RoboDK station: Example-01.a-Robot Painting - Universal Robots.rdk

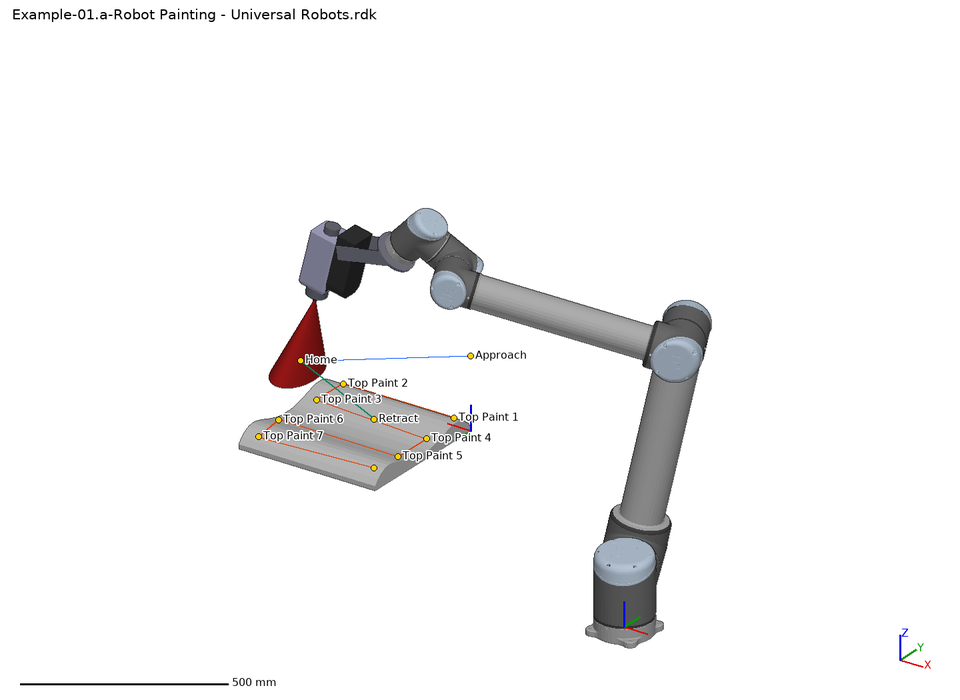
[picture v0: the station drawn from its stored meshes, robots at their saved joint values, targets as dots, program paths as lines]
Station Painting-Tutorial. Poses are relative to the parent item; angles as X-Y-Z fixed-axis rotations.
  - frame UR10 Base at (0, 0, 0) mm
    - robot UR10: 6 axes, payload 10 kg, reach 1300 mm, repeatability 0.1 mm, weight 28.9 kg
        modified DH rows (alpha deg, a mm, theta deg, d mm): 0, 0, 0, 118; 90, 0, 180, 0; 0, 612.7, 0, 0; 0, 571.6, 0, 163.9; -90, 0, 0, 115.7; 90, 0, 180, 92.2
        joint limits [-360, -360, -360, -360, -360, -360] to [360, 360, 360, 360, 360, 360]; home [0, -90, 90, 0, 90, 0]; saved at [-151.986, -78.222, -86.642, -64.602, 73.062, 110.032]
      - tool Paint gun, TCP at (50, 0, 450) mm, rotated rx 0 ry 30 rz 0 deg, size 203.2 x 279.7 x 471.5 mm
    - frame Frame 2 at (-800, 500, 100) mm, rotated rx 0 ry 0 rz 180 deg
      - object Object Inspection at (0, 0, 0) mm, size 400 x 400 x 46.2 mm, geometry from Object Inspection.stp
      - target Home (Cartesian target) at (66.76, 615.12, 413.71) mm, rotated rx 179.14 ry 13.35 rz -178.18 deg; joints [-151.986, -78.222, -86.642, -64.602, 73.062, 110.032] of UR10
      - target Approach (Cartesian target) at (0, 0, 200) mm, rotated rx 180 ry 0 rz 180 deg; joints [-208.691, -96.314, -82.153, -64.673, 103.889, 64.641] of UR10
      - target Top Paint 1 (Cartesian target) at (31.07, 24.78, 35.36) mm, rotated rx 143.81 ry -11.15 rz 165.19 deg; joints [-219.536, -114.993, -76.946, -70.137, 127.814, 81.267] of UR10
      - target Top Paint 2 (Cartesian target) at (355.2, 25.82, 36.15) mm, rotated rx 143.1 ry -8.02 rz 169.48 deg; joints [-210.289, -143.985, -30.818, -80.427, 128.618, 88.068] of UR10
      - target Top Paint 3 (Cartesian target) at (364.05, 124.58, 30.83) mm, rotated rx -163.01 ry 5.38 rz 162.95 deg; joints [-179.629, -118.486, -75.308, -44.885, 65.562, 96.641] of UR10
      - target Top Paint 4 (Cartesian target) at (29.88, 140.33, 26.47) mm, rotated rx -165.93 ry 6.07 rz 157.13 deg; joints [-177.894, -88.354, -112.979, -39.189, 64.009, 104.945] of UR10
      - target Top Paint 5 (Cartesian target) at (29.25, 262.96, 27.37) mm, rotated rx 165.04 ry -3.2 rz 168.19 deg; joints [-194.064, -91.552, -105.349, -45.917, 103.957, 95.559] of UR10
      - target Top Paint 6 (Cartesian target) at (379.27, 259.84, 26.52) mm, rotated rx 164.87 ry -2.25 rz 171.75 deg; joints [-190.188, -122.622, -65.046, -54.105, 103.992, 95.944] of UR10
      - target Top Paint 7 (Cartesian target) at (357.91, 376.6, 34.28) mm, rotated rx -142.62 ry 4.77 rz 173.79 deg; joints [-157.813, -118.488, -80.898, -50.291, 43.391, 100.711] of UR10
      - target Top Paint 8 (Cartesian target) at (25.99, 366.61, 39.82) mm, rotated rx -154.85 ry 4.87 rz 169.75 deg; joints [-153.215, -84.837, -115.212, -52.717, 50.654, 115.012] of UR10
      - target Retract (Cartesian target) at (25.99, 366.61, 169.82) mm, rotated rx -154.85 ry 4.87 rz 169.75 deg; joints [-153.215, -81.897, -104.364, -66.506, 50.654, 115.012] of UR10
  - program ApproachMove (4 instructions, listed below)
  - program PaintTop (11 instructions, listed below)
  - program Retract (4 instructions, listed below)
  - program MainProg (5 instructions, listed below)
  - Python program SprayOn (listed below)
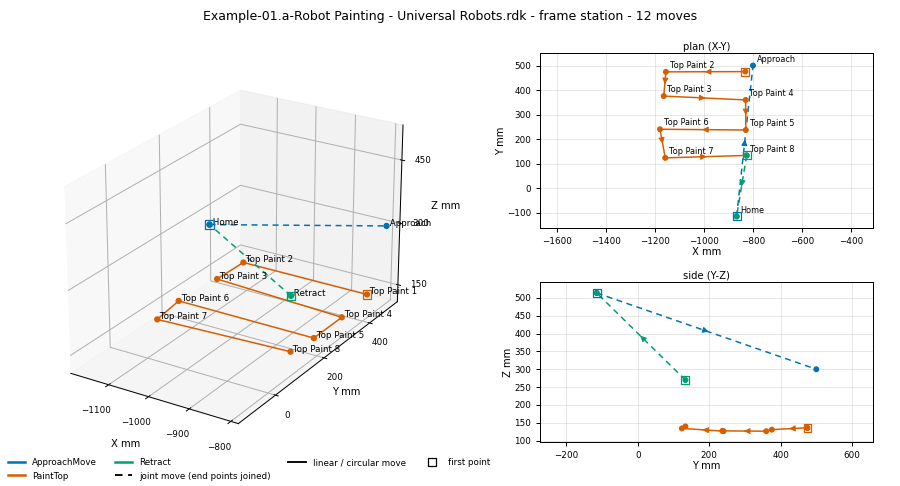
[picture p0: tool path of Example-01.a-Robot Painting - Universal Robots.rdk in frame station, 12 of 12 moves have a stored position in this frame; points joined in program order, loops and branches not executed]

--- program ApproachMove (robot UR10) ---
  Set Ref.: Frame 2
  Set Tool: Paint gun
  MoveJ (Home)
  MoveJ (Approach)

--- program PaintTop (robot UR10) ---
  Set Ref.: Frame 2
  Set Tool: Paint gun
  MoveJ (Top Paint 1)
  Set speed (50.0 mm/s)
  MoveL (Top Paint 2)
  MoveL (Top Paint 3)
  MoveL (Top Paint 4)
  MoveL (Top Paint 5)
  MoveL (Top Paint 6)
  MoveL (Top Paint 7)
  MoveL (Top Paint 8)

--- program Retract (robot UR10) ---
  Set Ref.: Frame 2
  Set Tool: Paint gun
  MoveL (Retract)
  MoveJ (Home)

--- program MainProg (robot UR10) ---
  Call ApproachMove
  Call SprayOn(1)
  Call PaintTop
  Call SprayOn(0)
  Call Retract

--- Python program SprayOn ---
# This macro allows simulating a spray gun
# It is possible to call SprayOn(1) to simulate turning the Spray gun ON or GunOn(0) to stop simulating the gun
# Calling SprayOn(-1) clears all displayed data
# The macro will output spray gun statistics

# For more information visit:
# http://www.robodk.com/doc/PythonAPI/robolink.html

# Define the default action (0 to deactivate, +1 to activate, -1 to clear any spray gun simulation)
# Setting it to None will display a message
ACTION = None

from robolink import *    # API to communicate with RoboDK
from robodk import *      # basic matrix operations
RDK = Robolink()

# quit if we are not in simulation mode
if RDK.RunMode() != RUNMODE_SIMULATE:
    quit()

# Get any previously added spray gun simulations and display statistics (spray on the part vs spray falling out of the part)
info, data = RDK.Spray_GetStats()
if data.size(1) > 0:
    print("Spray gun statistics:")
    print(info)
    print(data.tr())
    # # Diplay statistics
    # RDK.ShowMessage("Material used: %.1f%%<br>Material waisted: %.1f%%<br>Total particles: %.1f" % (data[1,0],data[2,0],data[3,0]), True)
    # # Clear previous spray
    # RDK.Spray_Clear()

# Check if we are running this program inside another program and passing arguments
import sys
if len(sys.argv) > 1:
    ACTION = int(sys.argv[1])

# If the default ACTION is None, display a message to activate/deactivate the spray gun
if ACTION is None:
    print('Note: This macro can be called as GunOn(1) or GunOn(0)')
    entry = mbox('Turn gun ON or OFF', ('On', '1'), ('Off', '0'))
    if not entry:
        quit()
    ACTION = int(entry)

if ACTION == 0:
    # Turn the gun off
    RDK.Spray_SetState(SPRAY_OFF)

if ACTION < 0:
    # Clear all spray simulations
    RDK.Spray_Clear()

elif ACTION > 0:
    # Create a new spray gun object in RoboDK
    # by using RDK.Spray_Add(tool, object, options_command, volume, geometry)
    # tool: tool item (TCP) to use
    # object: object to project the particles
    # options_command (optional): string to specify options. Example:
    #     STEP=AxB: Defines the grid to be projected 1x1 means only one line of particle projection (for example, for welding)
    #     PARTICLE: Defines the shape and size of particle (sphere or particle), unless a specific geometry is provided:
    #       a- SPHERE(radius, facets)
    #       b- SPHERE(radius, facets, scalex, scaley, scalez)
    #       b- CUBE(sizex, sizey, sizez)
    #     RAND=factor: Defines a random factor factor 0 means that the particles are not deposited randomly
    #     ELLYPSE: defines the volume as an ellypse (default)
    #     RECTANGLE: defines the volume as a rectangle
    #     PROJECT: project the particles to the surface (default) (for welding, painting or scanning)
    #     NO_PROJECT: does not project the particles to the surface (for example, for 3D printing)
    #
    # volume (optional): Matrix of parameters defining the volume of the spray gun
    # geometry (optional): Matrix of vertices defining the triangles.


    tool = 0    # auto detect active tool
    obj = 0     # auto detect object in active reference frame
    # We can specify a given tool object and/or object
    #robot = RDK.Item("ABB IRB 2600-12/1.85", ITEM_TYPE_ROBOT)
    #tools = robot.Childs()
    #if len(tools) > 0:
    #    tool = tools[0]
    #obj = RDK.Item('object', ITEM_TYPE_OBJECT)

    options_command = "ELLYPSE PROJECT PARTICLE=SPHERE(4,8,1,1,0.5) STEP=8x8 RAND=2" # simulate
    #options_command = "PARTICLE=CUBE(10,10,2) STEP=8x8"
    #options_command = "PARTICLE=SPHERE(4,8) STEP=8x8"
    #options_command = "PARTICLE=SPHERE(4,8,1,1,0.1) STEP=8x8 RAND=3"

    # Example commands for welding:
    # options_command = "PROJECT PARTICLE=SPHERE(4,8)"
    # options_command = PARTICLE=SPHERE(4,8) STEP=1x0


    # define the ellypse volume as p0, pA, pB, colorRGBA (close and far), in mm
    # coordinates must be provided with respect to the TCP
    close_p0 = [   0,   0, -200] # xyz in mm
    close_pA = [   5,   0, -200] # xyz in mm
    close_pB = [   0,  10, -200] # xyz in mm
    close_color = [ 1, 0, 0, 1]  # RGBA (0-1)

    far_p0   = [   0,   0,  50] # xyz in mm
    far_pA   = [  60,   0,  50] # xyz in mm
    far_pB   = [   0, 120,  50] # xyz in mm
    far_color   = [ 0, 0, 1, 0.2]  # RGBA (0-1)

    close_param = close_p0 + close_pA + close_pB + close_color
    far_param = far_p0 + far_pA + far_pB + far_color
    volume = Mat([close_param, far_param]).tr()
    RDK.Spray_Add(tool, obj, options_command, volume)
    RDK.Spray_SetState(SPRAY_ON)


    # Another example with a varying rectancular shape
    # define the rectangular volume as p0, pA, pB, colorRGBA (close and far)
    # close_param = [-90,-117,  0,  90,-117,0,   -90,117,  0,       0.2,0.2,1,.1]
    # far_param   = [-175,-190,200, 175,-190,200,   -175,190,200,   0.5,0,0,.9]
    # volume = Mat([close_param, far_param])
    # RDK.Spray_Add(tool, obj, "RECTANGLE PARTICLE=SPHERE(2,5) STEP=15x15 RAND=3", volume.tr())
    # RDK.Spray_SetState(SPRAY_ON)

    # Optional: define geometry as a list of triangles with normals (instead of a scaled cube or a sphere)
    # geom = Mat([[0,0,0,   0,0,1], [5,0,0,   0,0,1], [0,5,0,   0,0,1]])
    # RDK.Spray_Add(tool, obj, "STEP=8x8 RANDX=3", volume.tr(), geom.tr())
    # RDK.Spray_SetState(SPRAY_ON)
